ABB RAPID module: Wobj_base_nest_legs_2.mod

MODULE Wobj_base_nest_legs_2
	! Points are read in order of declaration.
  ! Please do not change the order of points!

  LOCAL PERS robtarget pWobj_U_PointX1:=[[1226.434,71.38622,-447.0584],[0.00202518329024315,-0.520143866539001,-0.854075372219086,0.00122601550538093],[0,0,0,0],[9E+09,9E+09,9E+09,9E+09,9E+09,9E+09]];
	LOCAL PERS robtarget pWobj_U_PointX2:=[[653.2594,-588.1196,-462.8528],[0.00208390178158879,-0.520320236682892,-0.853967845439911,0.00120840640738606],[-1,-1,0,0],[9E+09,9E+09,9E+09,9E+09,9E+09,9E+09]];
	LOCAL PERS robtarget pWobj_U_PointY1:=[[1693.002,-334.7816,-449.3624],[0.193330451846123,0.961640179157257,-0.189692303538322,-0.0434553287923336],[-1,-1,2,0],[9E+09,9E+09,9E+09,9E+09,9E+09,9E+09]];

ENDMODULE
